(****************************************************************************************)
(*							Beckhoff Automation Poland									*)
(*								FB_SaveTextToFile  v1.0									*)
(*									26.06.2014											*)
(* Blok funkcyjny zapisujacy tekst do pliku, maksymalna dlugosc wpisu 1000 znakow		*)
(*______________________________________________________________________________________*)
FUNCTION_BLOCK FB_SaveTextToFile
VAR_INPUT
	bExecute		: BOOL;			(* Komenda wpisu *)
	AmsNetId		: T_AmsNetId;	(* AMS NET ID obiektu docelowego, gdy lokalnie, to zmienna moze byc pusta *)
	sPath			: STRING; 		(* Sciezka pliku, np  'Hard Disk\'*)
	sName			: STRING; 		(* Nazwa pliku wraz z rozszerzeniem 'LogFile.txt'; *)
	sLine			: STRING(1000);	(* Tresc wpisu *)
END_VAR
VAR_OUTPUT
	bBusy: 			BOOL;
	bError: 		BOOL;
END_VAR
VAR
	fbFileOpen: 	FB_FileOpen;
	ftOpen: 		F_TRIG;
	fbFilePuts: 	FB_FilePutText;
	ftPuts: 		F_TRIG;
	fbFileClose:	FB_FileClose;
	ftClose: 		F_TRIG;
END_VAR
VAR // added by the converter: edge detectors and wires of the graphical bodies
    _w1 : BOOL;
END_VAR

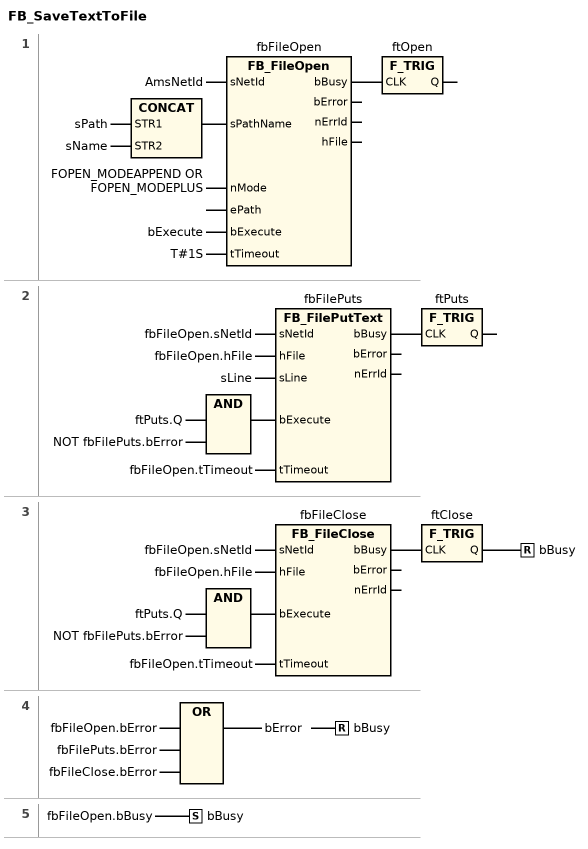
// NETWORK 1
fbFileOpen(
    sNetId := AmsNetId,
    sPathName := CONCAT(STR1 := sPath, STR2 := sName),
    nMode := FOPEN_MODEAPPEND OR FOPEN_MODEPLUS,
    bExecute := bExecute,
    tTimeout := T#1S); // FB_FileOpen
ftOpen(CLK := fbFileOpen.bBusy); // F_TRIG

// NETWORK 2
fbFilePuts(
    sNetId := fbFileOpen.sNetId,
    hFile := fbFileOpen.hFile,
    sLine := sLine,
    bExecute := ftPuts.Q AND (NOT fbFilePuts.bError),
    tTimeout := fbFileOpen.tTimeout); // FB_FilePutText
ftPuts(CLK := fbFilePuts.bBusy); // F_TRIG

// NETWORK 3
fbFileClose(
    sNetId := fbFileOpen.sNetId,
    hFile := fbFileOpen.hFile,
    bExecute := ftPuts.Q AND (NOT fbFilePuts.bError),
    tTimeout := fbFileOpen.tTimeout); // FB_FileClose
ftClose(CLK := fbFileClose.bBusy); // F_TRIG
bBusy R= ftClose.Q;

// NETWORK 4
_w1 := fbFileOpen.bError OR fbFilePuts.bError OR fbFileClose.bError;
bError := _w1;
bBusy R= _w1;

// NETWORK 5
bBusy S= fbFileOpen.bBusy;

END_FUNCTION_BLOCK

(* stored: Version 1.1.0.1, ProductVersion 3.1.4026.13, FileIdentifier 5ba757791692c25c1a62ec816c0826299281d853, FileSignature 2b70b14cab307a7fa37b8a61a959369e85b6388b05cd5068da05fc06f1de1c91de71866d593f21a7e3d19d8c58758ad1fbf8b27dd259adfdc4ef4b5e9d4a7f30c75952140132097e4877ddfd54c6a4a18903ea9b831c70766da2fce9e2e8920190095e7536cf4b12e8c54dbd5751d3adb6857fae7983f53538f51ccc7bf9b709ed0168cd3e23883ab606cc8cdfffca0368339e6f256128b8fc22a7e4aab0287ddafd957cc45bbef4cc9c72d2e8750d14dcf3ae16b1a667b2d248be46f6f3222a0b4e29ca2a86af204bdd06dac0313cfdb295f8a773382e6a13bddc96edb9a853c405a7e00bcd31e2a32fa5f70b6dda2c2f470b9ea0b14ab2a95f9e7cfaaa2abc
   POU FB_SaveTextToFile: Id {c05d2e28-4203-4212-81e8-60e87bf4526e}, SpecialFunc None *)
